// TwinCAT 3 PLC project Movement
// ProgramVersion: 3.1.4023.0
// libraries:
//   TcUnit, * (www.tcunit.org)
// project tree:
//   / POU_Test.TcPOU
//   TwoPointMovement/ FB_Position.TcPOU, FB_SimpleLinearTwoWayDrive.TcPOU, FB_TwoWayPneumaticDrive.TcPOU, IPosition.TcIO, ITwoPointMovement.TcIO
//   TwoPointMovement/Test/ FB_SimpleLinearTwoWayDrive_Test.TcPOU

// ---- TwoPointMovement/IPosition.TcIO
INTERFACE IPosition

METHOD Lock : BOOL
VAR_INPUT
END_VAR
END_METHOD

PROPERTY Locked : BOOL
GET
END_GET
END_PROPERTY

METHOD MoveTo : BOOL
VAR_INPUT
END_VAR
END_METHOD

PROPERTY Moving : BOOL
GET
END_GET
END_PROPERTY

PROPERTY Reached : BOOL
GET
END_GET
END_PROPERTY

END_INTERFACE

// ---- TwoPointMovement/ITwoPointMovement.TcIO
INTERFACE ITwoPointMovement

PROPERTY InHomePos : BOOL
GET
END_GET
END_PROPERTY

PROPERTY InWorkPos : BOOL
GET
END_GET
END_PROPERTY

METHOD ToHomePos : BOOL
VAR_INPUT
END_VAR
END_METHOD

METHOD ToWorkPos : BOOL
VAR_INPUT
END_VAR
END_METHOD

END_INTERFACE

// ---- POU_Test.TcPOU
PROGRAM POU_Test
VAR
	fbSimpleLinearTwoWayDriveTest: FB_SimpleLinearTwoWayDrive_Test;
END_VAR

TcUnit.RUN();

END_PROGRAM

// ---- TwoPointMovement/Test/FB_SimpleLinearTwoWayDrive_Test.TcPOU
FUNCTION_BLOCK FB_SimpleLinearTwoWayDrive_Test EXTENDS FB_TestSuite
VAR_INPUT
END_VAR
VAR_OUTPUT
END_VAR
VAR
END_VAR

METHOD No_Movement_When_Locked : BOOL
VAR_INPUT
END_VAR
VAR
	sut: FB_SimpleLinearTwoWayDrive;
END_VAR
TEST('No movement should be possible when locked');

sut(
	SensorHomePos := TRUE,
	SensorWorkPos := FALSE,
	Enable := FALSE,
	ToHome := FALSE,
	ToWork := FALSE);
	
AssertEquals(FALSE, sut.ActorWorkPos, 'Movement even if not enabled');

TEST_FINISHED();
END_METHOD

END_FUNCTION_BLOCK

// ---- TwoPointMovement/FB_SimpleLinearTwoWayDrive.TcPOU
FUNCTION_BLOCK FB_SimpleLinearTwoWayDrive
VAR_INPUT
	SensorHomePos: BOOL;
	SensorWorkPos: BOOL;
	Enable: BOOL;
	ToHome: BOOL;
	ToWork: BOOL;
END_VAR
VAR_OUTPUT
	ActorHomePos: BOOL;
	ActorWorkPos: BOOL;
END_VAR
VAR
END_VAR

ActorHomePos := Enable AND ToHome AND NOT ActorWorkPos AND NOT SensorHomePos;
ActorWorkPos := Enable AND ToWork AND NOT ActorHomePos AND NOT SensorWorkPos;

END_FUNCTION_BLOCK

// ---- TwoPointMovement/FB_Position.TcPOU
FUNCTION_BLOCK FB_Position IMPLEMENTS IPosition
VAR_INPUT
	Sensor: BOOL;
END_VAR
VAR_OUTPUT
	Actor: BOOL;
END_VAR
VAR
END_VAR

// Release Signal
Locked := FALSE;

{warning 'Methodenimplementierung hinzufügen'}
METHOD Lock : BOOL
Locked := TRUE;
END_METHOD

PROPERTY Locked : BOOL
GET
VAR_INST
	_locked: BOOL;
END_VAR
END_GET
END_PROPERTY

METHOD MoveTo : BOOL
Actor := NOT Reached AND NOT Locked;
END_METHOD

PROPERTY Moving : BOOL
GET
Moving := Actor;
END_GET
END_PROPERTY

PROPERTY Reached : BOOL
GET
Reached := Sensor;
END_GET
END_PROPERTY

END_FUNCTION_BLOCK

// ---- TwoPointMovement/FB_TwoWayPneumaticDrive.TcPOU
FUNCTION_BLOCK FB_TwoWayPneumaticDrive IMPLEMENTS ITwoPointMovement
VAR_INPUT
END_VAR
VAR_OUTPUT
END_VAR
VAR
END_VAR

{warning 'Eigenschaftenimplementierung hinzufügen'}
PROPERTY InHomePos : BOOL
GET
END_GET
END_PROPERTY

{warning 'Eigenschaftenimplementierung hinzufügen'}
PROPERTY InWorkPos : BOOL
GET
END_GET
END_PROPERTY

{warning 'Methodenimplementierung hinzufügen'}
METHOD ToHomePos : BOOL
END_METHOD

{warning 'Methodenimplementierung hinzufügen'}
METHOD ToWorkPos : BOOL
END_METHOD

END_FUNCTION_BLOCK
